// LS Electric XG5000 project: fdsafa
// PLC NewPLC
// module base 0 slot 0: 입출력 모듈:XBC-DR32H (DC 24V 입력, 릴레이 출력 32점)

PROGRAM NewProgram (task: 스캔 프로그램)

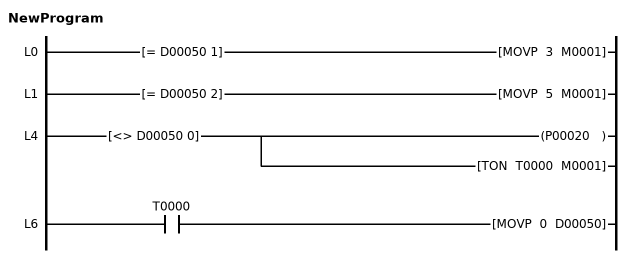
; L0
LOAD=     D00050 1
MOVP      3 M0001
; L1
LOAD=     D00050 2
MOVP      5 M0001
; L4
LOAD<>    D00050 0
OUT       P00020
TON       T0000 M0001
; L6
LOAD      T0000
MOVP      0 D00050